TYPE DigitalInputBase_50022E7B :
STRUCT
END_STRUCT
END_TYPE

(* stored: Version 1.1.0.1, ProductVersion 3.1.4024.9
   DUT DigitalInputBase_50022E7B: Id {151b47c0-d881-0152-31c7-434ce319c490} *)
